FUNCTION_BLOCK FB_CellCheckPart_Test EXTENDS TcUnit.FB_TestSuite
VAR
END_VAR

CheckPartGood();
CheckPartBadBarcode();

METHOD PRIVATE CheckPartBadBarcode
VAR
	fbCell		: FB_Cell;
	MockStatus	: ST_PartStatus;
	Expected	: BOOL := FALSE;
	Result		: BOOL;
END_VAR
MockStatus.bBarcodeStatus := FALSE;
MockStatus.bCapperStatus := TRUE;
MockStatus.bFillerStatus := TRUE;
MockStatus.bWeightStatus := TRUE;

Result := fbCell.CheckPart(MockStatus);

AssertEquals(Expected := Expected,
             Actual := Result,
             Message := 'part check mismatch');

TEST_FINISHED();
END_METHOD

METHOD PRIVATE CheckPartGood
VAR
	fbCell		: FB_Cell;
	MockStatus	: ST_PartStatus;
	Expected	: BOOL := TRUE;
	Result		: BOOL;
END_VAR
MockStatus.bBarcodeStatus := TRUE;
MockStatus.bCapperStatus := TRUE;
MockStatus.bFillerStatus := TRUE;
MockStatus.bWeightStatus := TRUE;

Result := fbCell.CheckPart(MockStatus);

AssertEquals(Expected := Expected,
             Actual := Result,
             Message := 'part check mismatch');

TEST_FINISHED();
END_METHOD

END_FUNCTION_BLOCK

(* stored: Version 1.1.0.1, ProductVersion 3.1.4024.12
   POU FB_CellCheckPart_Test: Id {5d8408a8-2a16-4833-8353-0d244cf7fe20}, SpecialFunc None
   Method CheckPartBadBarcode: Id {00ac122f-4718-41a9-beea-3eb9fb4aba3b}
   Method CheckPartGood: Id {4589c4d3-6f4d-4ca9-850a-ce7aa2ca1fe6} *)
